Yaskawa INFORM job: MASTER_X4.JBI

/JOB
//NAME MASTER_X4
///FOLDERNAME MASTER_ODWLOK
//POS
///NPOS 90,90,90,0,0,0
///TOOL 0
///POSTYPE PULSE
///PULSE
C00000=2000,-113621,-91819,0,89172,0
///TOOL 1
C00001=12644,-114998,-116551,5579,58951,81855
///TOOL 0
C00002=3161,-91504,-85468,2682,88050,79011
C00003=3161,-91504,-85468,2682,88050,79011
///TOOL 1
C00004=12644,-114998,-116551,5579,58951,81855
///TOOL 0
C00005=32835,-100330,-111373,-6266,63391,89303
///TOOL 1
C00006=12644,-114998,-116551,5579,58951,81855
///TOOL 0
C00007=26539,-106348,-113568,-2696,61319,87093
C00008=25079,-107553,-113996,-1846,60923,86561
C00009=12644,-114998,-116551,5579,58951,81855
///TOOL 1
C00010=12644,-114998,-116551,5579,58951,81855
///TOOL 0
C00011=3643,-76224,-106676,19950,71810,76872
///TOOL 1
C00012=12644,-114998,-116551,5579,58951,81855
C00013=12644,-114998,-116551,5579,58951,81855
C00014=12644,-114998,-116551,5579,58951,81855
C00015=12644,-114998,-116551,5579,58951,81855
///TOOL 0
C00016=12644,-114998,-116551,5579,58951,81855
///TOOL 1
C00017=-118839,-50376,-74715,5087,87435,-13721
///TOOL 0
C00018=-84515,-86778,-73230,-5241,65800,-2317
///TOOL 1
C00019=12644,-114998,-116551,5579,58951,81855
///TOOL 0
C00020=3643,-76224,-106676,19950,71810,76872
///TOOL 1
C00021=12644,-114998,-116551,5579,58951,81855
C00022=12644,-114998,-116551,5579,58951,81855
C00023=12644,-114998,-116551,5579,58951,81855
C00024=12644,-114998,-116551,5579,58951,81855
C00025=12644,-114998,-116551,5579,58951,81855
C00026=12644,-114998,-116551,5579,58951,81855
C00027=12644,-114998,-116551,5579,58951,81855
C00028=12644,-114998,-116551,5579,58951,81855
///TOOL 0
C00029=-159584,-34280,-73725,-5274,106726,39066
C00030=-147283,4412,-21796,10805,51416,45079
C00031=-126083,-46964,-66593,-7674,58401,55640
C00032=-71874,-146793,-98010,-56220,44659,85303
///TOOL 1
C00033=12644,-114998,-116551,5579,58951,81855
///TOOL 0
C00034=3643,-76224,-106676,19950,71810,76872
///TOOL 1
C00035=12644,-114998,-116551,5579,58951,81855
///TOOL 0
C00036=12644,-114998,-116551,5579,58951,81855
///TOOL 1
C00037=12644,-114998,-116551,5579,58951,81855
///TOOL 0
C00038=12644,-114998,-116551,5579,58951,81855
C00039=12644,-114998,-116551,5579,58951,81855
C00040=-36470,-76528,-106815,19279,71473,77234
C00041=-35459,-77320,-107015,18997,71215,77329
C00042=-34937,-74855,-105907,18653,71663,77576
C00043=-34937,-74855,-105907,18653,71663,77576
///TOOL 1
C00044=12644,-114998,-116551,5579,58951,81855
C00045=12644,-114998,-116551,5579,58951,81855
C00046=12644,-114998,-116551,5579,58951,81855
///TOOL 0
C00047=3643,-76224,-106676,19950,71810,76872
C00048=12644,-114998,-116551,5579,58951,81855
C00049=-103618,-56678,-54869,-17247,39327,-49180
C00050=-92545,-86083,-73453,-28460,38949,-42906
///TOOL 1
C00051=12644,-114998,-116551,5579,58951,81855
///TOOL 0
C00052=12644,-114998,-116551,5579,58951,81855
///TOOL 1
C00053=12644,-114998,-116551,5579,58951,81855
///TOOL 0
C00054=12644,-114998,-116551,5579,58951,81855
C00055=12644,-114998,-116551,5579,58951,81855
C00056=-9037,-143537,-113247,5913,77526,79136
C00057=12432,-115277,-116519,5582,59133,81828
///TOOL 1
C00058=12644,-114998,-116551,5579,58951,81855
C00059=12644,-114998,-116551,5579,58951,81855
///TOOL 0
C00060=12644,-114998,-116551,5579,58951,81855
///TOOL 1
C00061=12644,-114998,-116551,5579,58951,81855
C00062=12644,-114998,-116551,5579,58951,81855
C00063=12644,-114998,-116551,5579,58951,81855
///TOOL 0
C00064=-107750,-95748,-53471,-77151,35098,40175
C00065=-122924,45358,33156,-57774,46766,29048
///TOOL 1
C00066=12644,-114998,-116551,5579,58951,81855
C00067=12644,-114998,-116551,5579,58951,81855
///TOOL 0
C00068=-160592,-79427,-90579,66425,81632,-32083
///TOOL 1
C00069=12644,-114998,-116551,5579,58951,81855
C00070=12644,-114998,-116551,5579,58951,81855
C00071=12644,-114998,-116551,5579,58951,81855
C00072=12644,-114998,-116551,5579,58951,81855
///TOOL 0
C00073=12644,-114998,-116551,5579,58951,81855
///TOOL 1
C00074=12644,-114998,-116551,5579,58951,81855
C00075=12644,-114998,-116551,5579,58951,81855
C00076=12644,-114998,-116551,5579,58951,81855
C00077=12644,-114998,-116551,5579,58951,81855
///TOOL 0
C00078=5980,-86291,-109240,16219,68472,78166
C00079=5980,-86291,-109240,16219,68472,78166
///TOOL 1
C00080=12644,-114998,-116551,5579,58951,81855
///TOOL 0
C00081=12644,-114998,-116551,5579,58951,81855
C00082=12644,-114998,-116551,5579,58951,81855
C00083=12644,-114998,-116551,5579,58951,81855
C00084=12644,-114998,-116551,5579,58951,81855
C00085=12644,-114998,-116551,5579,58951,81855
C00086=12644,-114998,-116551,5579,58951,81855
C00087=-51438,-141397,-114999,40946,67363,37514
C00088=-51438,-141397,-114999,40946,67363,37514
C00089=2000,-113618,-91816,15,89172,1
BC00000=87189,670739,720296
BC00001=204899,680330,1075141
BC00002=87842,675035,1040975
BC00003=87842,675035,1040975
BC00004=204899,680330,1075141
BC00005=204899,706161,1075141
BC00006=204899,680330,1075141
BC00007=204899,697628,1075141
BC00008=204899,695724,1075141
BC00009=204899,680330,1075141
BC00010=204899,680330,1075141
BC00011=199464,674570,1075173
BC00012=204899,680330,1075141
BC00013=204899,680330,1075141
BC00014=204899,680330,1075141
BC00015=204899,680330,1075141
BC00016=204899,680330,1075141
BC00017=300252,736283,216702
BC00018=222140,708483,216702
BC00019=204899,680330,1075141
BC00020=199464,674570,1075173
BC00021=204899,680330,1075141
BC00022=204899,680330,1075141
BC00023=204899,680330,1075141
BC00024=204899,680330,1075141
BC00025=204899,680330,1075141
BC00026=204899,680330,1075141
BC00027=204899,680330,1075141
BC00028=204899,680330,1075141
BC00029=218952,814745,125477
BC00030=218952,684872,125477
BC00031=202221,684872,125477
BC00032=167027,684872,125477
BC00033=204899,680330,1075141
BC00034=199464,674570,1075173
BC00035=204899,680330,1075141
BC00036=204899,680330,1075141
BC00037=204899,680330,1075141
BC00038=204899,680330,1075141
BC00039=204899,680330,1075141
BC00040=295325,674563,1075175
BC00041=293463,674682,1075174
BC00042=293463,674682,1075174
BC00043=293463,674682,1075174
BC00044=204899,680330,1075141
BC00045=204899,680330,1075141
BC00046=204899,680330,1075141
BC00047=199464,674570,1075173
BC00048=204899,680330,1075141
BC00049=106862,754848,165353
BC00050=106862,672256,165353
BC00051=204899,680330,1075141
BC00052=204899,682250,1075141
BC00053=204899,680330,1075141
BC00054=204899,680330,1075141
BC00055=204899,680330,1075141
BC00056=324407,673965,978757
BC00057=206069,680268,1074197
BC00058=204899,680330,1075141
BC00059=204899,680330,1075141
BC00060=204899,680330,1075141
BC00061=204899,680330,1075141
BC00062=204899,680330,1075141
BC00063=204899,680330,1075141
BC00064=144630,673121,681655
BC00065=144630,814605,366796
BC00066=204899,680330,1075141
BC00067=204899,680330,1075141
BC00068=315224,676573,283186
BC00069=204899,680330,1075141
BC00070=204899,680330,1075141
BC00071=204899,680330,1075141
BC00072=204899,680330,1075141
BC00073=204899,680330,1075141
BC00074=204899,680330,1075141
BC00075=204899,680330,1075141
BC00076=204899,680330,1075141
BC00077=204899,680330,1075141
BC00078=197437,676065,1075165
BC00079=197437,676065,1075165
BC00080=204899,680330,1075141
BC00081=204899,680330,1075141
BC00082=204899,680330,1075141
BC00083=204899,680330,1075141
BC00084=204899,680330,1075141
BC00085=204899,680330,1075141
BC00086=204899,680330,1075141
BC00087=157489,678871,1075149
BC00088=157489,678871,1075149
BC00089=87190,687250,596160
EC00000=0,0
EC00001=0,0
EC00002=0,1112952
EC00003=0,0
EC00004=-798156,0
EC00005=-798156,1112951
EC00006=-860235,803798
EC00007=-860235,309153
EC00008=-798156,0
EC00009=-317951,1051120
EC00010=399078,61830
EC00011=798156,0
EC00012=798156,0
EC00013=266052,92745
EC00014=266052,1020205
EC00015=798156,1112951
EC00016=798156,1112951
EC00017=798156,1112951
EC00018=798156,1112951
EC00019=798156,1112951
EC00020=-798156,1112951
EC00021=-798156,0
EC00022=-221710,154576
EC00023=221710,958374
EC00024=798156,1112951
EC00025=798156,1112951
EC00026=266052,1020205
EC00027=266052,92745
EC00028=798156,0
EC00029=798156,0
EC00030=798156,0
EC00031=798156,0
EC00032=798156,0
EC00033=487762,0
EC00034=-454111,-556475
EC00035=1596313,-556475
EC00036=1596313,-556475
EC00037=1596313,-556475
EC00038=1595260,12593
EC00039=1595260,12593
EC00040=-1418945,-556475
EC00041=-1418932,1112951
EC00042=798156,1112951
EC00043=798156,1112951
EC00044=798156,1112951
EC00045=266052,1020205
EC00046=266052,92745
EC00047=798156,0
EC00048=798156,0
EC00049=798156,0
EC00050=798156,0
EC00051=798156,0
EC00052=798156,0
EC00053=798156,0
EC00054=798156,0
EC00055=-1373963,0
EC00056=21022,556477
EC00057=790546,556475
EC00058=798156,556475
EC00059=0,556475
EC00060=0,556475
EC00061=0,556475
EC00062=310394,1112951
EC00063=798156,1112951
EC00064=798156,1112951
EC00065=798156,1112951
EC00066=-798156,1112951
EC00067=798156,0
EC00068=798156,0
EC00069=798156,0
EC00070=1463287,0
EC00071=1418945,-556475
EC00072=1330261,-556475
EC00073=1330261,-556475
EC00074=1330261,-556475
EC00075=1596313,556475
EC00076=1596313,556475
EC00077=1862365,0
EC00078=348771,296
EC00079=348771,554591
EC00080=798156,556475
EC00081=517805,556475
EC00082=335055,861512
EC00083=335055,1089512
EC00084=335055,1089512
EC00085=335055,861512
EC00086=517805,556475
EC00087=346849,306373
EC00088=347217,1384
EC00089=1,0
//INST
///DATE 2025/03/17 12:02
///ATTR SC,RW
///GROUP1 RB1,BS1
///GROUP2 ST1
NOP
WAIT IG#(285)=255
CLEAR B060 1
COMM DOUT OT#(1433) ON
DOUT OT#(1435) ON
MOVJ C00000 BC00000 VJ=100.00  +MOVJ EC00000 VJ=100.00
MOVJ C00001 BC00001 VJ=100.00  +MOVJ EC00001 VJ=100.00
CALL JOB:KRIS1A
MOVJ C00002 BC00002 VJ=100.00  +MOVJ EC00002 VJ=100.00
MOVJ C00003 BC00003 VJ=100.00  +MOVJ EC00003 VJ=100.00
MOVJ C00004 BC00004 VJ=100.00  +MOVJ EC00004 VJ=100.00
CALL JOB:CLEAN-R1_KM_3P
'-90,0
CALL JOB:OK_R2_O242(-90,180)OKKR
'-90,180
MOVJ C00005 BC00005 VJ=100.00  +MOVJ EC00005 VJ=100.00
MOVJ C00006 BC00006 VJ=100.00  +MOVJ EC00006 VJ=100.00
MOVJ C00007 BC00007 VJ=100.00  +MOVJ EC00007 VJ=100.00
MOVJ C00008 BC00008 VJ=100.00  +MOVJ EC00008 VJ=100.00
CALL JOB:CLEAN-R1_KM_3P
'-90,0
CALL JOB:OK_R2_O6-7(-90,0)OKKR
'-90,180
MOVJ C00009 BC00009 VJ=100.00  +MOVJ EC00009 VJ=100.00
MOVJ C00010 BC00010 VJ=100.00  +MOVJ EC00010 VJ=100.00
MOVJ C00011 BC00011 VJ=100.00  +MOVJ EC00011 VJ=100.00
CALL JOB:CLEAN-R1_KM_3P
'90,0
CALL JOB:OK_R2_O8A-O21A(90,0)OKKR
'90,0
MOVJ C00012 BC00012 VJ=100.00  +MOVJ EC00012 VJ=100.00
MOVJ C00013 BC00013 VJ=100.00  +MOVJ EC00013 VJ=100.00
MOVJ C00014 BC00014 VJ=100.00  +MOVJ EC00014 VJ=100.00
MOVJ C00015 BC00015 VJ=100.00  +MOVJ EC00015 VJ=100.00
CALL JOB:CLEAN-R1_KM_3P
MOVJ C00016 BC00016 VJ=100.00  +MOVJ EC00016 VJ=100.00
'90,180
CALL JOB:OK_R2_O8B-O21B(90,0)_MPKMOK
MOVJ C00017 BC00017 VJ=100.00  +MOVJ EC00017 VJ=100.00
MOVJ C00018 BC00018 VJ=100.00  +MOVJ EC00018 VJ=100.00
'90,180
MOVJ C00019 BC00019 VJ=100.00  +MOVJ EC00019 VJ=100.00
MOVJ C00020 BC00020 VJ=100.00  +MOVJ EC00020 VJ=100.00
CALL JOB:CLEAN-R1_KM_3P
'-90,180
CALL JOB:OK_R2_O22-23(-90,180)OKKR
'-90,0
MOVJ C00021 BC00021 VJ=100.00  +MOVJ EC00021 VJ=100.00
MOVJ C00022 BC00022 VJ=100.00  +MOVJ EC00022 VJ=100.00
MOVJ C00023 BC00023 VJ=100.00  +MOVJ EC00023 VJ=100.00
MOVJ C00024 BC00024 VJ=100.00  +MOVJ EC00024 VJ=100.00
CALL JOB:CLEAN-R1_KM_3P
'90,180
CALL JOB:OK_R2_O24A(90,180)OKKR
'90,180
MOVJ C00025 BC00025 VJ=100.00  +MOVJ EC00025 VJ=100.00
CALL JOB:CLEAN-R1_KM_3P
MOVJ C00026 BC00026 VJ=100.00  +MOVJ EC00026 VJ=100.00
MOVJ C00027 BC00027 VJ=100.00  +MOVJ EC00027 VJ=100.00
MOVJ C00028 BC00028 VJ=100.00  +MOVJ EC00028 VJ=100.00
'90,0
CALL JOB:OK_R2_O24B(90,0)KMOK
MOVJ C00029 BC00029 VJ=100.00  +MOVJ EC00029 VJ=100.00
MOVJ C00030 BC00030 VJ=100.00  +MOVJ EC00030 VJ=100.00
MOVJ C00031 BC00031 VJ=100.00  +MOVJ EC00031 VJ=100.00
MOVJ C00032 BC00032 VJ=100.00  +MOVJ EC00032 VJ=100.00
'90,0
MOVJ C00033 BC00033 VJ=100.00  +MOVJ EC00033 VJ=100.00
MOVJ C00034 BC00034 VJ=100.00  +MOVJ EC00034 VJ=100.00
CALL JOB:CLEAN-R1_KM_3P
'-60,-90
CALL JOB:OK_R2_O27-28(-60,-90)OKKR
'-60,-90
MOVJ C00035 BC00035 VJ=100.00  +MOVJ EC00035 VJ=100.00
CALL JOB:CLEAN-R1_KM_3P
MOVJ C00036 BC00036 VJ=100.00  +MOVJ EC00036 VJ=100.00
'180,-90
CALL JOB:OK_R2_O7,1(180,-90)OKKR_COMOUT
'180,-90
MOVJ C00037 BC00037 VJ=100.00  +MOVJ EC00037 VJ=100.00
MOVJ C00038 BC00038 VJ=100.00  +MOVJ EC00038 VJ=100.00
CALL JOB:CLEAN-R1_KM_3P
MOVJ C00039 BC00039 VJ=100.00  +MOVJ EC00039 VJ=100.00
'180,50
CALL JOB:KRIS1(-160_-90)07
CALL JOB:CLEAN-R1_KM_3P
CALL JOB:KRIS2(-160_-90)34
MOVJ C00040 BC00040 VJ=100.00  +MOVJ EC00040 VJ=100.00
MOVJ C00041 BC00041 VJ=100.00  +MOVJ EC00041 VJ=100.00
MOVJ C00042 BC00042 VJ=100.00  +MOVJ EC00042 VJ=100.00
CALL JOB:CLEAN-R1_KM_3P
MOVJ C00043 BC00043 VJ=100.00  +MOVJ EC00043 VJ=100.00
'90,180
CALL JOB:OK_R2_O38-47,64(1)(90,180)OKKR
'90,180
MOVJ C00044 BC00044 VJ=100.00  +MOVJ EC00044 VJ=100.00
MOVJ C00045 BC00045 VJ=100.00  +MOVJ EC00045 VJ=100.00
MOVJ C00046 BC00046 VJ=100.00  +MOVJ EC00046 VJ=100.00
MOVJ C00047 BC00047 VJ=100.00  +MOVJ EC00047 VJ=100.00
CALL JOB:CLEAN-R1_KM_3P
MOVJ C00048 BC00048 VJ=100.00  +MOVJ EC00048 VJ=100.00
'90,0
CALL JOB:OK_R2_O38-47,64(2)(90,0)_MPOK
MOVJ C00049 BC00049 VJ=100.00  +MOVJ EC00049 VJ=100.00
MOVJ C00050 BC00050 VJ=100.00  +MOVJ EC00050 VJ=100.00
'90,0
MOVJ C00051 BC00051 VJ=100.00  +MOVJ EC00051 VJ=100.00
CALL JOB:CLEAN-R1_KM_3P
MOVJ C00052 BC00052 VJ=100.00  +MOVJ EC00052 VJ=100.00
'90,0
CALL JOB:OK_R2_O50&56(110_90,0)AWOK
'90,0
MOVJ C00053 BC00053 VJ=100.00  +MOVJ EC00053 VJ=100.00
CALL JOB:CLEAN-R1_KM_3P
MOVJ C00054 BC00054 VJ=100.00  +MOVJ EC00054 VJ=100.00
MOVJ C00055 BC00055 VJ=100.00  +MOVJ EC00055 VJ=100.00
CALL JOB:KRIS3(-160_-90)54
CALL JOB:KRIS4(-224_-90)
CALL JOB:KRIS5(-224_-90)
'180,50
MOVJ C00056 BC00056 VJ=99.00  +MOVJ EC00056 VJ=100.00
MOVJ C00057 BC00057 VJ=99.00  +MOVJ EC00057 VJ=99.00
CALL JOB:CLEAN-R1_KM_3P
'90,90
CALL JOB:OK_R2_O54(90,90)AWOK
'90,90
'!!!!!!!!!!!!!!!!!!
PAUSE
'JUDASZ
'VIKTOR
'WYMIEN KONCOWKE PRADOWA
'!!!!!!!!!!!!!!!!!!
MOVJ C00058 BC00058 VJ=100.00  +MOVJ EC00058 VJ=100.00
MOVJ C00059 BC00059 VJ=100.00  +MOVJ EC00059 VJ=100.00
CALL JOB:CLEAN-R1_KM_3P
MOVJ C00060 BC00060 VJ=100.00  +MOVJ EC00060 VJ=100.00
CALL JOB:KRIS6(-12_90)
'0,90
MOVJ C00061 BC00061 VJ=100.00  +MOVJ EC00061 VJ=100.00
MOVJ C00062 BC00062 VJ=100.00  +MOVJ EC00062 VJ=100.00
MOVJ C00063 BC00063 VJ=100.00  +MOVJ EC00063 VJ=100.00
CALL JOB:CLEAN-R1_KM_3P
'90,180
MOVJ C00064 BC00064 VJ=100.00  +MOVJ EC00064 VJ=100.00
MOVJ C00065 BC00065 VJ=100.00  +MOVJ EC00065 VJ=100.00
CALL JOB:OK_R2_O57-69(2)(90,0)_OK
'90,180
CALL JOB:CLEAN-R1_KM_3P
MOVJ C00066 BC00066 VJ=100.00  +MOVJ EC00066 VJ=100.00
'-90,180
CALL JOB:OK_R2_O29-32(90,0_180)OKKR
'-90,0
MOVJ C00067 BC00067 VJ=100.00  +MOVJ EC00067 VJ=100.00
CALL JOB:CLEAN-R1_KM_3P
'90,0
MOVJ C00068 BC00068 VJ=100.00  +MOVJ EC00068 VJ=100.00
CALL JOB:OK_R2_O57-69(1)(90,0)_OK
'90,0
MOVJ C00069 BC00069 VJ=100.00  +MOVJ EC00069 VJ=100.00
MOVJ C00070 BC00070 VJ=100.00  +MOVJ EC00070 VJ=100.00
MOVJ C00071 BC00071 VJ=100.00  +MOVJ EC00071 VJ=100.00
MOVJ C00072 BC00072 VJ=100.00  +MOVJ EC00072 VJ=100.00
CALL JOB:CLEAN-R1_KM_3P
MOVJ C00073 BC00073 VJ=100.00  +MOVJ EC00073 VJ=10.00
'150,-90
CALL JOB:OK_R2_O48(150,-90)AWOK
'150,-90
MOVJ C00074 BC00074 VJ=100.00  +MOVJ EC00074 VJ=100.00
MOVJ C00075 BC00075 VJ=100.00  +MOVJ EC00075 VJ=100.00
CALL JOB:CLEAN-R1_KM_3P
'180,90
CALL JOB:OK_R2_O49(180,90)AWOK
'180,90
'SPRAWDZIC PRZEJAZD
MOVJ C00076 BC00076 VJ=100.00  +MOVJ EC00076 VJ=100.00
MOVJ C00077 BC00077 VJ=100.00  +MOVJ EC00077 VJ=100.00
CALL JOB:CLEAN-R1_KM_3P
CALL JOB:X4-SCHODKI_ZEW
CALL JOB:CLEAN-R1_KM_3P
MOVJ C00078 BC00078 VJ=100.00  +MOVJ EC00078 VJ=100.00
MOVJ C00079 BC00079 VJ=100.00  +MOVJ EC00079 VJ=100.00
'90,90
CALL JOB:OK_R2_O25(90,90)OKKR
'90,90
MOVJ C00080 BC00080 VJ=100.00  +MOVJ EC00080 VJ=100.00
MOVJ C00081 BC00081 VJ=100.00  +MOVJ EC00081 VJ=100.00
MOVJ C00082 BC00082 VJ=100.00  +MOVJ EC00082 VJ=100.00
MOVJ C00083 BC00083 VJ=100.00  +MOVJ EC00083 VJ=100.00
CALL JOB:OK_R2_O55A(90,180)KMOK
MOVJ C00084 BC00084 VJ=100.00  +MOVJ EC00084 VJ=100.00
MOVJ C00085 BC00085 VJ=100.00  +MOVJ EC00085 VJ=100.00
MOVJ C00086 BC00086 VJ=100.00  +MOVJ EC00086 VJ=100.00
MOVJ C00087 BC00087 VJ=100.00  +MOVJ EC00087 VJ=100.00
MOVJ C00088 BC00088 VJ=100.00  +MOVJ EC00088 VJ=100.00
CALL JOB:OK_R2_O55B(90,0)KMOK
CALL JOB:KRIS_OTHER_WELDS
CALL JOB:KRIS7(1)_V2
CALL JOB:KRIS7_V2
COMM CALL JOB:KRIS7
'zmiana KRIS7 na KRIS7(1)_V2
'oraz KRIS7_V2
CALL JOB:CLEAN-R1_KM_3P
CALL JOB:N_R2_D50&56B(110_90,180)
MOVJ C00089 BC00089 VJ=100.00  +MOVJ EC00089 VJ=100.00
COMM DOUT OT#(1433) OFF
DOUT OT#(1435) OFF
PAUSE
PAUSE
ABORT
PAUSE
END
